// TIA Portal V20 export
// export: Created 2025-09-14T10:59:00.0000000Z, ExportSetting WithDefaults
VAR_GLOBAL   // PLC tag table "TagTable_DO"
   RTU1_SF_StartCmd AT %Q0.0 : Bool;
   RTU1_C_Comp1Cmd AT %Q0.1 : Bool;
   RTU1_H_Heat1Cmd AT %Q0.2 : Bool;
END_VAR
